FUNCTION F_ColorToStringHexColor : STRING
VAR_INPUT
	color : UDINT;
END_VAR

IF color = STATICS.stColor.None THEN
	F_ColorToStringHexColor := STATICS.stColor.NoneString;
ELSIF color = STATICS.stColor.Transparent THEN
	F_ColorToStringHexColor := STATICS.stColor.TransparentString;	
ELSIF color = STATICS.stColor.Theme THEN
	F_ColorToStringHexColor := STATICS.stColor.ThemeString;
ELSE
	F_ColorToStringHexColor  := Concat(
								'#',
								Delete(
									DWORD_TO_HEXSTR(
											color,
											8,
											FALSE)
									,2
									,1));//#hexadecimal
END_IF

END_FUNCTION

(* stored: Version 1.1.0.1, ProductVersion 3.1.4024.12
   POU F_ColorToStringHexColor: Id {1e1b512c-5673-4d7e-946d-c71c1048e02b}, SpecialFunc None *)
